(* CODESYS project tcl_unittestlibrary.library
   Company: Red Rock Controls Limited
   Description: Initial Release
   Version: 1.0.0.0
   Placeholder: tcl_UnitTestLibrary
   Author: Roger Christopher
   Title: tcl_UnitTestLibrary

Project tree, tasks and I/O mapping:
  libraries: Tc2_Standard, * (Beckhoff Automation GmbH); Tc2_System, * (Beckhoff Automation GmbH); Tc2_Utilities, * (Beckhoff Automation GmbH); Tc3_Module, * (Beckhoff Automation GmbH); tcl_StringUtils, * (Red Rock Controls Limited); Tc3_DynamicMemory, * (Beckhoff Automation GmbH)
  DUTs/
    data type ST_TestResult
  Functions/
  GVLs/
    global variables Parameters
  Unit Test Framework/
    Assertions/
      function block T_Assertion [ST]: Assert, AssertEquals_BLOB, AssertEquals_BOOL, AssertEquals_BYTE, AssertEquals_DINT, AssertEquals_DWORD, AssertEquals_INT, AssertEquals_INTERFACE, AssertEquals_LINT, AssertEquals_LREAL, AssertEquals_PVOID, AssertEquals_REAL, AssertEquals_STRING, AssertEquals_UDINT, AssertEquals_UINT, AssertEquals_ULINT, AssertEquals_WORD, AssertNotEquals_INTERFACE, AssertionFailed, AssertionMessage
    List Of Tests/
      interface I_ListOfTests: Count, GetTest
      function block T_ListOfTests [ST]: AddTest, Clear, Count, FB_exit, FB_init, GetTest
      function block T_TestIterator [ST]: FB_init, GetNext, HasMore, Reset
    Test Runner/
      function block T_TestRunner [ST]: AddTest, Execute, FB_init, Initialise
    Unit Test/
      function F_LogResult [ST]
      interface I_UnitTest: FailMessage, Init, Run, TestCompleted, TestFailed, TestName
      function block T_UnitTestBase [ST]: CheckAssertion, FailMessage, FB_init, Init, Run, SetTestName, TestCompleted, TestFailed, TestName
  Version/
    global variables Global_Version
*)

// DUTs/ST_TestResult
TYPE
    ST_TestResult :
    STRUCT
        TestCompleted : BOOL;
        TestFailed    : BOOL;
        FailMessage   : T_MaxString;
    END_STRUCT
END_TYPE

// GVLs/Parameters
VAR_GLOBAL CONSTANT
    MAX_TESTS : DINT := 200;
END_VAR

// Version/Global_Version
{attribute 'TcGenerated'}
{attribute 'no-analysis'}
{attribute 'linkalways'}
// This function has been automatically generated from the project information.
VAR_GLOBAL CONSTANT
    {attribute 'const_non_replaced'}
    stLibVersion_tcl_UnitTestLibrary : ST_LibVersion := (iMajor    := 1,
                                                         iMinor    := 0,
                                                         iBuild    := 0,
                                                         iRevision := 0,
                                                         nFlags    := 0,
                                                         sVersion  := '1.0.0.0');
END_VAR

// Unit Test Framework/Assertions/T_Assertion
FUNCTION_BLOCK T_Assertion
VAR_INPUT
END_VAR
VAR_OUTPUT
END_VAR
VAR
    _AssertionFailed  : BOOL;
    _AssertionMessage : T_MaxString;
    _ExpectedAsString : T_MaxString;
    _ActualAsString   : T_MaxString;
END_VAR

METHOD Assert
VAR_INPUT
    Caller           : T_MaxString;
    AssertionMessage : T_MaxString;
    Expected         : T_MaxString;
    Actual           : T_MaxString;
END_VAR
_AssertionFailed  := TRUE;
_AssertionMessage := F_FormatStringEx2('Assertion failed in %s - %s', Caller, AssertionMessage);
_ExpectedAsString := F_FormatStringEx1('  Expected = %s', Expected);
_ActualAsString   := F_FormatStringEx1('  Actual   = %s', Actual);
END_METHOD

METHOD AssertEquals_BLOB
VAR_INPUT
    Expected     : ANY;
    Actual       : ANY;
    VariableName : T_MaxString;
END_VAR
IF Expected.diSize <> Actual.diSize THEN
    _AssertionFailed  := TRUE;
    _AssertionMessage := F_FormatStringEx1('AssertEquals_BLOB failed in %s : Sizes differ', VariableName);

ELSIF Expected.TypeClass <> Actual.TypeClass THEN
    _AssertionFailed  := TRUE;
    _AssertionMessage := F_FormatStringEx1('AssertEquals_BLOB failed in %s: TypeClasses differ', VariableName);

ELSIF
    MEMCMP(pBuf1 := Expected.pValue, pBuf2 := Actual.pValue, n := DINT_TO_UDINT(Actual.diSize)) <> 0 THEN
    _AssertionFailed  := TRUE;
    _AssertionMessage := F_FormatStringEx1('AssertEquals_BLOB failed in %s: Contents differ', VariableName);
ELSE
    _AssertionFailed  := FALSE;
    _AssertionMessage := '';
END_IF
END_METHOD

METHOD AssertEquals_BOOL
VAR_INPUT
    Expected     : BOOL;
    Actual       : BOOL;
    VariableName : T_MaxString;
END_VAR
IF Expected <> Actual THEN
    _AssertionFailed  := TRUE;
    _AssertionMessage := F_FormatStringEx3('AssertEquals_BOOL failed : Variable "%s" =  %s, expected = %s', VariableName, BOOL_TO_STRING(Actual), BOOL_TO_STRING(Expected));
ELSE
    _AssertionFailed  := FALSE;
    _AssertionMessage := '';
END_IF
END_METHOD

METHOD AssertEquals_BYTE
VAR_INPUT
    Expected     : BYTE;
    Actual       : BYTE;
    VariableName : T_MaxString;
END_VAR
IF Expected <> Actual THEN
    _AssertionFailed  := TRUE;
    _AssertionMessage := F_FormatString3('AssertEquals_BYTE failed : Variable "%s" =  %d, expected = %d', F_STRING(VariableName), F_BYTE(Actual), F_BYTE(Expected));
ELSE
    _AssertionFailed  := FALSE;
    _AssertionMessage := '';
END_IF
END_METHOD

METHOD AssertEquals_DINT
VAR_INPUT
    Expected     : DINT;
    Actual       : DINT;
    VariableName : T_MaxString;
END_VAR
IF Expected <> Actual THEN
    _AssertionFailed  := TRUE;
    _AssertionMessage := F_FormatString3('AssertEquals_DINT failed : Variable "%s" =  %d, expected = %d', F_STRING(VariableName), F_DINT(Actual), F_DINT(Expected));
ELSE
    _AssertionFailed  := FALSE;
    _AssertionMessage := '';
END_IF
END_METHOD

METHOD AssertEquals_DWORD
VAR_INPUT
    Expected     : DWORD;
    Actual       : DWORD;
    VariableName : T_MaxString;
END_VAR
IF Expected <> Actual THEN
    _AssertionFailed  := TRUE;
    _AssertionMessage := F_FormatString3('AssertEquals_DWORD failed : Variable "%s" =  %d, expected = %d', F_STRING(VariableName), F_DWORD(Actual), F_DWORD(Expected));
ELSE
    _AssertionFailed  := FALSE;
    _AssertionMessage := '';
END_IF
END_METHOD

METHOD AssertEquals_INT
VAR_INPUT
    Expected     : INT;
    Actual       : INT;
    VariableName : T_MaxString;
END_VAR
IF Expected <> Actual THEN
    _AssertionFailed  := TRUE;
    _AssertionMessage := F_FormatString3('AssertEquals_INT failed : Variable "%s" =  %d, expected = %d', F_STRING(VariableName), F_INT(Actual), F_INT(Expected));
ELSE
    _AssertionFailed  := FALSE;
    _AssertionMessage := '';
END_IF
END_METHOD

METHOD AssertEquals_INTERFACE
VAR_INPUT
    Expected     : __SYSTEM.IQueryInterface;
    Actual       : __SYSTEM.IQueryInterface;
    VariableName : T_MaxString;
END_VAR
IF Expected <> Actual THEN
    _AssertionFailed  := TRUE;
    _AssertionMessage := F_FormatString1('AssertEquals_INTERFACE failed : Variable "%s"', F_STRING(VariableName));
ELSE
    _AssertionFailed  := FALSE;
    _AssertionMessage := '';
END_IF
END_METHOD

METHOD AssertEquals_LINT
VAR_INPUT
    Expected     : LINT;
    Actual       : LINT;
    VariableName : T_MaxString;
END_VAR
IF Expected <> Actual THEN
    _AssertionFailed  := TRUE;
    _AssertionMessage := F_FormatString3('AssertEquals_LINT failed : Variable "%s" =  %d, expected = %d', F_STRING(VariableName), F_LINT(Actual), F_LINT(Expected));
ELSE
    _AssertionFailed  := FALSE;
    _AssertionMessage := '';
END_IF
END_METHOD

METHOD AssertEquals_LREAL
VAR_INPUT
    Expected     : LREAL;
    Actual       : LREAL;
    Delta        : LREAL;
    VariableName : T_MaxString;
END_VAR
IF ABS(Expected - Actual) > Delta THEN
    _AssertionFailed  := TRUE;
    _AssertionMessage := F_FormatString3('AssertEquals_LREAL failed : Variable "%s" =  %f, expected = %f', F_STRING(VariableName), F_LREAL(Actual), F_LREAL(Expected));
ELSE
    _AssertionFailed  := FALSE;
    _AssertionMessage := '';
END_IF
END_METHOD

METHOD AssertEquals_PVOID
VAR_INPUT
    Expected     : PVOID;
    Actual       : PVOID;
    VariableName : T_MaxString;
END_VAR
IF Expected <> Actual THEN
    _AssertionFailed  := TRUE;
    _AssertionMessage := F_FormatString1('AssertEquals_PVOID failed : Variable "%s"', F_STRING(VariableName));
ELSE
    _AssertionFailed  := FALSE;
    _AssertionMessage := '';
END_IF
END_METHOD

METHOD AssertEquals_REAL
VAR_INPUT
    Expected     : REAL;
    Actual       : REAL;
    Delta        : REAL;
    VariableName : T_MaxString;
END_VAR
IF ABS(Expected - Actual) > Delta THEN
    _AssertionFailed  := TRUE;
    _AssertionMessage := F_FormatString3('AssertEquals_REAL failed : Variable "%s" =  %f, expected = %f', F_STRING(VariableName), F_REAL(Actual), F_REAL(Expected));
ELSE
    _AssertionFailed  := FALSE;
    _AssertionMessage := '';
END_IF
END_METHOD

METHOD AssertEquals_STRING
VAR_INPUT
    Expected     : T_MaxString;
    Actual       : T_MaxString;
    VariableName : T_MaxString;
END_VAR
IF Expected <> Actual THEN
    _AssertionFailed  := TRUE;
    _AssertionMessage := F_FormatString3('AssertEquals_STRING failed : Variable "%s" =  %s, expected = %s', F_STRING(VariableName), F_STRING(Actual), F_STRING(Expected));
ELSE
    _AssertionFailed  := FALSE;
    _AssertionMessage := '';
    _ExpectedAsString := '';
    _ActualAsString   := '';
END_IF
END_METHOD

METHOD AssertEquals_UDINT
VAR_INPUT
    Expected     : UDINT;
    Actual       : UDINT;
    VariableName : T_MaxString;
END_VAR
IF Expected <> Actual THEN
    _AssertionFailed  := TRUE;
    _AssertionMessage := F_FormatString3('AssertEquals_UDINT failed : Variable "%s" =  %d, expected = %d', F_STRING(VariableName), F_UDINT(Actual), F_UDINT(Expected));
ELSE
    _AssertionFailed  := FALSE;
    _AssertionMessage := '';
END_IF
END_METHOD

METHOD AssertEquals_UINT
VAR_INPUT
    Expected     : UINT;
    Actual       : UINT;
    VariableName : T_MaxString;
END_VAR
IF Expected <> Actual THEN
    _AssertionFailed  := TRUE;
    _AssertionMessage := F_FormatString3('AssertEquals_UINT failed : Variable "%s" =  %d, expected = %d', F_STRING(VariableName), F_UINT(Actual), F_UINT(Expected));
ELSE
    _AssertionFailed  := FALSE;
    _AssertionMessage := '';
END_IF
END_METHOD

METHOD AssertEquals_ULINT
VAR_INPUT
    Expected     : ULINT;
    Actual       : ULINT;
    VariableName : T_MaxString;
END_VAR
IF Expected <> Actual THEN
    _AssertionFailed  := TRUE;
    _AssertionMessage := F_FormatString3('AssertEquals_ULINT failed : Variable "%s" =  %d, expected = %d', F_STRING(VariableName), F_ULINT(Actual), F_ULINT(Expected));
ELSE
    _AssertionFailed  := FALSE;
    _AssertionMessage := '';
END_IF
END_METHOD

METHOD AssertEquals_WORD
VAR_INPUT
    Expected     : WORD;
    Actual       : WORD;
    VariableName : T_MaxString;
END_VAR
IF Expected <> Actual THEN
    _AssertionFailed  := TRUE;
    _AssertionMessage := F_FormatString3('AssertEquals_WORD failed : Variable "%s" =  %d, expected = %d', F_STRING(VariableName), F_WORD(Actual), F_WORD(Expected));
ELSE
    _AssertionFailed  := FALSE;
    _AssertionMessage := '';
END_IF
END_METHOD

METHOD AssertNotEquals_INTERFACE
VAR_INPUT
    Expected     : __SYSTEM.IQueryInterface;
    Actual       : __SYSTEM.IQueryInterface;
    VariableName : T_MaxString;
END_VAR
IF Expected = Actual THEN
    _AssertionFailed  := TRUE;
    _AssertionMessage := F_FormatString1('AssertNotEquals_INTERFACE failed : Variable "%s"', F_STRING(VariableName));
ELSE
    _AssertionFailed  := FALSE;
    _AssertionMessage := '';
END_IF
END_METHOD

PROPERTY AssertionFailed : BOOL
GET
AssertionFailed := _AssertionFailed;
END_GET
END_PROPERTY

PROPERTY AssertionMessage : T_MaxString
GET
AssertionMessage := _AssertionMessage;
END_GET
END_PROPERTY

END_FUNCTION_BLOCK

// Unit Test Framework/List Of Tests/I_ListOfTests
INTERFACE I_ListOfTests

PROPERTY Count : DINT
GET
END_GET
END_PROPERTY

METHOD GetTest : I_UnitTest
VAR_INPUT
    Index : DINT;
END_VAR
END_METHOD

END_INTERFACE

// Unit Test Framework/Unit Test/I_UnitTest
INTERFACE I_UnitTest EXTENDS __SYSTEM.IQueryInterface

PROPERTY FailMessage : T_MaxString;
GET
END_GET
END_PROPERTY

METHOD Init : BOOL
VAR_INPUT
END_VAR
END_METHOD

METHOD FINAL Run
END_METHOD

PROPERTY TestCompleted : BOOL
GET
END_GET
END_PROPERTY

PROPERTY TestFailed : BOOL
GET
END_GET
END_PROPERTY

PROPERTY TestName : T_MaxString
GET
END_GET
END_PROPERTY

END_INTERFACE

// Unit Test Framework/List Of Tests/T_ListOfTests
FUNCTION_BLOCK T_ListOfTests IMPLEMENTS I_ListOfTests
VAR
    Buffer               : FB_DynMem_Buffer(ipMemMan := DynamicMemoryManager);
    DynamicMemoryManager : FB_DynMem_Manager;
    pTest                : POINTER TO I_UnitTest;
    TestCount            : DINT;
    Capacity             : DINT;
END_VAR

METHOD AddTest
VAR_INPUT
    Test : I_UnitTest;
END_VAR
IF Count = Capacity THEN
    Capacity := Capacity * 2;
    Buffer.Resize(nSize     := DINT_TO_UDINT(Capacity) * SIZEOF(PVOID),
                  bPreserve := TRUE,
                  bReset    := FALSE);

    pTest := Buffer.pBuffer;
END_IF

pTest[TestCount] := Test;
TestCount        := TestCount + 1;
END_METHOD

METHOD Clear
VAR_INPUT
END_VAR
Buffer.Clear();
TestCount := 0;
END_METHOD

PROPERTY Count : DINT
GET
Count := TestCount;
END_GET
END_PROPERTY

METHOD FB_exit : BOOL
VAR_INPUT
    bInCopyCode : BOOL; // if TRUE, the exit method is called for exiting an instance that is copied afterwards (online change).
END_VAR
IF NOT bInCopyCode THEN
    Buffer.DeleteBuffer();
    pTest := 0;
END_IF
END_METHOD

METHOD FB_init : BOOL
VAR_INPUT
    bInitRetains : BOOL; // if TRUE, the retain variables are initialized (warm start / cold start)
    bInCopyCode  : BOOL; // if TRUE, the instance afterwards gets moved into the copy code (online change)
    Capacity     : DINT;
END_VAR
Buffer.CreateBuffer(nSize  := DINT_TO_UDINT(Capacity) * SIZEOF(PVOID),
                    bReset := TRUE);

pTest          := Buffer.pBuffer;
THIS^.Capacity := Capacity;
END_METHOD

METHOD GetTest : I_UnitTest
VAR_INPUT
    Index : DINT;
END_VAR
IF Index < TestCount AND Index >= 0 THEN
    GetTest := pTest[Index];
END_IF
END_METHOD

END_FUNCTION_BLOCK

// Unit Test Framework/List Of Tests/T_TestIterator
FUNCTION_BLOCK T_TestIterator
VAR_INPUT
END_VAR
VAR_OUTPUT
END_VAR
VAR
    List  : I_ListOfTests;
    Index : DINT;
END_VAR

METHOD FB_init : BOOL
VAR_INPUT
    bInitRetains : BOOL; // if TRUE, the retain variables are initialized (warm start / cold start)
    bInCopyCode  : BOOL; // if TRUE, the instance afterwards gets moved into the copy code (online change)
    List         : I_ListOfTests;
END_VAR
THIS^.List := List;
END_METHOD

METHOD GetNext : I_UnitTest
VAR_INPUT
END_VAR
IF HasMore() THEN
    GetNext := List.GetTest(Index);
    Index   := Index + 1;
END_IF
END_METHOD

METHOD HasMore : BOOL
VAR_INPUT
END_VAR
HasMore := Index < List.Count and List.Count > 0;
END_METHOD

METHOD Reset
VAR_INPUT
END_VAR
Index := 0;
END_METHOD

END_FUNCTION_BLOCK

// Unit Test Framework/Test Runner/T_TestRunner
FUNCTION_BLOCK T_TestRunner
VAR
    State : (
        Init,
        GetTest,
        RunTest,
        CheckResults
    );
    TestGroupName    : T_MaxString;
    ResultsSummary   : T_MaxString;
    PassedTestsCount : DINT;
    FailedTestsCount : DINT;
    TestList         : T_ListOfTests(Capacity := 50);
    TestIterator     : T_TestIterator(TestList);
    CurrentTest      : I_UnitTest;
END_VAR

CASE State OF
    Init:
    // Wait for Execute();

    GetTest:
        IF TestIterator.HasMore() THEN
            CurrentTest := TestIterator.GetNext();
            State       := RunTest;
        ELSE
            CurrentTest := 0;
            State       := CheckResults;
        END_IF

    RunTest:
        CurrentTest.Run();

        IF CurrentTest.TestCompleted THEN
            IF CurrentTest.TestFailed THEN
                F_LogResult(Source := TestGroupName, Message := F_FormatStringEx2('Test Failed - %s (%s)', CurrentTest.TestName, CurrentTest.FailMessage));
                FailedTestsCount := FailedTestsCount + 1;
            ELSE
                F_LogResult(Source := TestGroupName, Message := F_FormatStringEx1('Test Passed - %s', CurrentTest.TestName));
                PassedTestsCount := PassedTestsCount + 1;
            END_IF

            State := GetTest;
        END_IF

    CheckResults:
        ResultsSummary := F_FormatString2('%d Tests Passed, %d Tests Failed',
                                          F_DINT(PassedTestsCount),
                                          F_DINT(FailedTestsCount));

        F_LogResult(Source := TestGroupName, Message := ResultsSummary);
        State := Init;

END_CASE

METHOD AddTest
VAR_INPUT
    UnitTest : I_UnitTest;
END_VAR
TestList.AddTest(UnitTest);
;
END_METHOD

METHOD Execute
VAR_INPUT
END_VAR
State := GetTest;
END_METHOD

METHOD FB_init : BOOL
VAR_INPUT
    bInitRetains  : BOOL; // if TRUE, the retain variables are initialized (warm start / cold start)
    bInCopyCode   : BOOL; // if TRUE, the instance afterwards gets moved into the copy code (online change)
    TestGroupName : T_MaxString;
END_VAR
THIS^.TestGroupName := TestGroupName;
END_METHOD

METHOD Initialise
VAR_INPUT
END_VAR
VAR
    i : DINT;
END_VAR
TestList.Clear();
TestIterator.Reset();

ResultsSummary   := '';
FailedTestsCount := 0;
PassedTestsCount := 0;
END_METHOD

END_FUNCTION_BLOCK

// Unit Test Framework/Unit Test/F_LogResult
FUNCTION F_LogResult : BOOL
VAR_INPUT
    Source  : T_MaxString;
    Message : T_MaxString;
END_VAR
VAR
END_VAR

ADSLOGSTR(msgCtrlMask := ADSLOG_MSGTYPE_STRING OR ADSLOG_MSGTYPE_ERROR OR ADSLOG_MSGTYPE_LOG,
          msgFmtStr   := F_FormatStringEx2('%s : %s', Source, Message),
          strArg      := '');

END_FUNCTION

// Unit Test Framework/Unit Test/T_UnitTestBase
{attribute 'reflection'}
{attribute 'hide_all_locals'}
FUNCTION_BLOCK T_UnitTestBase IMPLEMENTS I_UnitTest
VAR_INPUT
END_VAR
VAR_OUTPUT
END_VAR
VAR
    {attribute 'instance-path'}
    {attribute 'no_init'}
    _InstanceName : T_MaxString; // Automatically initialised with the full name of the instance
    _TestName     : T_MaxString;
    _TestResult   : ST_TestResult;

    Assertion : T_Assertion;
    State     : INT; // for general use during test...
END_VAR

METHOD CheckAssertion
VAR_INPUT
    NextState : INT;
END_VAR
IF Assertion.AssertionFailed THEN
    _TestResult.TestFailed    := TRUE;
    _TestResult.FailMessage   := Assertion.AssertionMessage;
    State                     := 0;
ELSE
    State := NextState;
END_IF

IF State = 0 THEN // we must be done...
	_TestResult.TestCompleted := TRUE;
END_IF
END_METHOD

PROPERTY FailMessage : T_MaxString;
GET
FailMessage := _TestResult.FailMessage;
END_GET
END_PROPERTY

METHOD FB_init : BOOL
VAR_INPUT
    bInitRetains : BOOL; // if TRUE, the retain variables are initialized (warm start / cold start)
    bInCopyCode  : BOOL; // if TRUE, the instance afterwards gets moved into the copy code (online change)
END_VAR
IF NOT bInCopyCode THEN // not an online change...
    THIS^.SetTestName();
END_IF
END_METHOD

METHOD Init : BOOL
_TestResult.TestFailed    := TRUE;
_TestResult.TestCompleted := FALSE;
_TestResult.FailMessage   := '';
State                     := 0;
END_METHOD

METHOD FINAL Run
THIS^();
END_METHOD

METHOD SetTestName
VAR
    StringSplitter : T_StringSplitter;
END_VAR
StringSplitter.Init(Str    := _InstanceName,
                    Delim1 := '.',
                    Delim2 := '');

WHILE StringSplitter.HasMore() DO
    _TestName := StringSplitter.GetNext(); // to get last sub-section
END_WHILE
END_METHOD

PROPERTY TestCompleted : BOOL
GET
TestCompleted := _TestResult.TestCompleted;
END_GET
END_PROPERTY

PROPERTY TestFailed : BOOL
GET
TestFailed := _TestResult.TestFailed;
END_GET
END_PROPERTY

PROPERTY TestName : T_MaxString
GET
TestName := _TestName;
END_GET
END_PROPERTY

END_FUNCTION_BLOCK
